		IF NOT fbEcSoERead.bError THEN
			(* read drive diagnostic *)
			fbEcSoERead(
				sNetId		:= stDriveRef.sNetId,
				nSlaveAddr	:= stDriveRef.nSlaveAddr,
				nIdn		:= 375,
				nElement	:= EC_SOE_ELEMENT_VALUE,
				nDriveNo	:= stDriveRef.nDriveNo,
				bCommand	:= FALSE,
				pDstBuf		:= piDiagNumber,
				cbBufLen	:= iSize,
				bExecute	:= FALSE,
				tTimeout	:= tTimeout
			);
			fbEcSoERead(bExecute := TRUE);
			iState	:= 20;
		ELSE
			bBusy	:= FALSE;
			bError	:= TRUE;
			iErrId	:= fbEcSoERead.nErrId;
			MEMSET(piDiagNumber, 0, iSize);
			dwAttribute := 0;
			iState	:= 0;
		END_IF
	END_IF

20: (* wait for read drive diag done *)
	fbEcSoERead(bExecute := FALSE);

	IF NOT fbEcSoERead.bBusy THEN
		fbEcSoERead(bExecute := FALSE);
		iState	:= 0;

		IF NOT fbEcSoERead.bError THEN
			bBusy	:= FALSE;
			(* clear remaining part of array *)
			IF (piDiagNumber^.iActualSize/4 < (iSize-4)/4 ) AND (piDiagNumber^.iMaxSize/4) = (iSize-4)/4 THEN
				FOR I := piDiagNumber^.iActualSize/4 TO (piDiagNumber^.iMaxSize/4) - 1 DO
					piDiagNumber^.arrDiagNumbers[I] := 0;
				END_FOR
			END_IF
		ELSE
			bBusy	:= FALSE;
			bError	:= TRUE;
			iErrId	:= fbEcSoERead.nErrId;
			MEMSET(piDiagNumber, 0, iSize);
		END_IF
	END_IF

END_CASE

bExecute_I := bExecute_I AND bExecute;
END_FUNCTION_BLOCK

(* POU FB_SoEReadMotorTemperature_ByDriveRef, ST *)
FUNCTION_BLOCK FB_SoEReadMotorTemperature_ByDriveRef
VAR_INPUT
	stDriveRef			: ST_DriveRef; 	(* contains sNetID of EcMaster, nSlaveAddr of EcDrive, nDriveNo of EcDrive, either preset or read from NC *)
	bExecute			: BOOL;				(* Function block execution is triggered by a rising edge at this input.*)
	tTimeout			: TIME := DEFAULT_ADS_TIMEOUT;(* States the time before the function is cancelled. *)
END_VAR
VAR_OUTPUT
	bBusy				: BOOL;
	bError				: BOOL;
	iAdsErrId			: UINT;
	iSercosErrId		: UINT;
	dwAttribute			: DWORD;
	fMotorTemperature	: REAL;
END_VAR
{library private}
VAR
	fbEcSoERead 		: FB_EcSoERead;
	iState				: INT;
	bExecute_I			: BOOL;
	iErrId				: UDINT;
	dwData				: ARRAY [0..1] OF DWORD;
	iMotorTemperature	: DINT;
	uiMotorTemperature	: UDINT;

	nFactor				: UINT;					(* bits  0..15 *)
	eLength				: E_SoE_AttribLen;		(* bits 16..18 *)
	eType				: E_SoE_Type;			(* bits 20..22 *)
	nComma				: USINT;				(* bits 24..27 *)
END_VAR
CASE iState OF
0: (* idle *)
	IF bExecute AND NOT bExecute_I THEN
		bExecute_I := bExecute;

		IF NOT bSeqReadDrvAttrAndValue THEN
			(* read Motor Temperature *)
			fbEcSoERead(
				sNetId		:= stDriveRef.sNetId,
				nSlaveAddr	:= stDriveRef.nSlaveAddr,
				nIdn		:= 383,
				nElement	:= 16#44, (* EC_SOE_ELEMENT_VALUE | EC_SOE_ELEMENT_ATTRIBUTE *)
				nDriveNo	:= stDriveRef.nDriveNo,
				bCommand	:= FALSE,
				pDstBuf		:= ADR(dwData),
				cbBufLen	:= SIZEOF(dwData),
				bExecute	:= FALSE,
				tTimeout	:= tTimeout
			);
			iState	:= 10;
		ELSE
			(* read attribute and Motor Temperature sequentially *)
			fbEcSoERead(
				sNetId		:= stDriveRef.sNetId,
				nSlaveAddr	:= stDriveRef.nSlaveAddr,
				nIdn		:= 383,
				nElement	:= EC_SOE_ELEMENT_ATTRIBUTE,
				nDriveNo	:= stDriveRef.nDriveNo,
				bCommand	:= FALSE,
				pDstBuf		:= ADR(dwData[0]),
				cbBufLen	:= SIZEOF(dwData[0]),
				bExecute	:= FALSE,
				tTimeout	:= tTimeout
			);
			iState	:= 5;
		END_IF
		fbEcSoERead(bExecute := TRUE);

		bBusy	:= TRUE;
		bError	:= FALSE;
		iErrId	:= 0;
		iAdsErrId		:= 0;
		iSercosErrId	:= 0;
	END_IF

5: (* wait for read Motor Temperature done *)
	fbEcSoERead(bExecute := FALSE);

	IF NOT fbEcSoERead.bBusy THEN
		fbEcSoERead(bExecute := FALSE);

		IF NOT fbEcSoERead.bError THEN
			(* read attribute and Motor Temperature sequentially *)
			fbEcSoERead(
				sNetId		:= stDriveRef.sNetId,
				nSlaveAddr	:= stDriveRef.nSlaveAddr,
				nIdn		:= 383,
				nElement	:= EC_SOE_ELEMENT_VALUE,
				nDriveNo	:= stDriveRef.nDriveNo,
				bCommand	:= FALSE,
				pDstBuf		:= ADR(dwData[1]),
				cbBufLen	:= SIZEOF(dwData[1]),
				bExecute	:= FALSE,
				tTimeout	:= tTimeout
			);
			fbEcSoERead(bExecute := TRUE);
			iState	:= 10;
		ELSE
			bBusy	:= FALSE;
			bError	:= TRUE;
			iErrId	:= fbEcSoERead.nErrId;
			iAdsErrId		:= UDINT_TO_UINT(iErrId);
			iSercosErrId	:= DWORD_TO_UINT(SHR((UDINT_TO_DWORD(iErrId) AND 16#FFFF0000),16));
			fMotorTemperature := 0;
			iState	:= 0;
		END_IF
	END_IF

10: (* wait for read Motor Temperature done *)
	fbEcSoERead(bExecute := FALSE);

	IF NOT fbEcSoERead.bBusy THEN
		fbEcSoERead(bExecute := FALSE);
		iState	:= 0;

		IF NOT fbEcSoERead.bError THEN
			bBusy	:= FALSE;
			dwAttribute := dwData[0];
			IF (dwAttribute <> 0) THEN
				nFactor	:= DWORD_TO_UINT(dwAttribute          AND 16#0000FFFF); (* bits  0..15 *)
				eLength	:= DWORD_TO_INT(SHR(dwAttribute,  16) AND 16#00000007);	(* bits 16..18 *)
				eType	:= DWORD_TO_INT(SHR(dwAttribute,  20) AND 16#00000007);	(* bits 20..22 *)
				nComma	:= DWORD_TO_USINT(SHR(dwAttribute,24) AND 16#0000000F); (* bits 24..27 *)
			END_IF

			CASE eType OF
			eSoE_Type_UNSIGNED, eSoE_Type_BIN, eSoE_Type_HEX:
				CASE eLength OF
					eSoE_LEN_2BYTE:
						uiMotorTemperature := 0;
						MEMCPY(ADR(uiMotorTemperature), ADR(dwData[1]), UDINT#2);
						fMotorTemperature := UDINT_TO_REAL(uiMotorTemperature) * nFactor / EXPT(10,nComma);
					eSoE_LEN_4BYTE:
						MEMCPY(ADR(uiMotorTemperature), ADR(dwData[1]), UDINT#4);
						fMotorTemperature := UDINT_TO_REAL(uiMotorTemperature) * nFactor / EXPT(10,nComma);
					ELSE
						bError := TRUE;
						iErrId := 16#705; (* parameter size not correct *)
						fMotorTemperature := 0;
				END_CASE

			eSoE_Type_SIGNED:
				CASE eLength OF
					eSoE_LEN_2BYTE:
						iMotorTemperature := 0;
						MEMCPY(ADR(iMotorTemperature), ADR(dwData[1]), UDINT#2);
						fMotorTemperature := DINT_TO_REAL(iMotorTemperature) * nFactor / EXPT(10,nComma);
					eSoE_LEN_4BYTE:
						MEMCPY(ADR(iMotorTemperature), ADR(dwData[1]), UDINT#4);
						fMotorTemperature := DINT_TO_REAL(iMotorTemperature) * nFactor / EXPT(10,nComma);
					ELSE
						bError := TRUE;
						iErrId := 16#705; (* parameter size not correct *)
						fMotorTemperature := 0;
				END_CASE

			ELSE
				bError := TRUE;
				iErrId := 16#706; (* invalid parameter value(s) *)
				fMotorTemperature := 0;
			END_CASE
		ELSE
			bBusy	:= FALSE;
			bError	:= TRUE;
			iErrId	:= fbEcSoERead.nErrId;
			iAdsErrId		:= UDINT_TO_UINT(iErrId);
			iSercosErrId	:= DWORD_TO_UINT(SHR((UDINT_TO_DWORD(iErrId) AND 16#FFFF0000),16));
			fMotorTemperature := 0;
		END_IF
	END_IF

END_CASE

bExecute_I := bExecute_I AND bExecute;
END_FUNCTION_BLOCK

(* POU FB_SoEReset_ByDriveRef, ST *)
FUNCTION_BLOCK FB_SoEReset_ByDriveRef
VAR_INPUT
	stDriveRef		: ST_DriveRef; 	(* contains sNetID of EcMaster, nSlaveAddr of EcDrive, nDriveNo of EcDrive, either preset or read from NC *)
	bExecute		: BOOL;			(* Function block execution is triggered by a rising edge at this input.*)
	tTimeout		: TIME := T#10s;(* States the time before the function is cancelled. (up to 10s) *)
END_VAR
VAR_OUTPUT
	bBusy			: BOOL;
	bError			: BOOL;
	iAdsErrId		: UINT;
	iSercosErrId	: UINT;
END_VAR
{library private}
VAR
	fbEcExecuteCmd	: FB_SoEExecuteCommand_ByDriveRef;
	iState			: INT;
	bExecute_I		: BOOL;
	iReset			: UINT := 3;
END_VAR
CASE iState OF
0: (* idle *)
	IF bExecute AND NOT bExecute_I THEN
		bExecute_I := bExecute;

		(* reset drive *)
		fbEcExecuteCmd(
			stDriveRef	:= stDriveRef,
			nIdn		:= S_0_IDN + 99,
			bExecute	:= FALSE,
			tTimeout	:= tTimeout
		);

		fbEcExecuteCmd(bExecute := TRUE);

		iState	:= 10;
		bBusy	:= TRUE;
		bError	:= FALSE;
		iAdsErrId		:= 0;
		iSercosErrId	:= 0;
	END_IF

10: (* wait for drive reset done *)
	fbEcExecuteCmd(bExecute := FALSE);

	IF NOT fbEcExecuteCmd.bBusy THEN
		fbEcExecuteCmd(bExecute := FALSE);

		IF NOT fbEcExecuteCmd.bError THEN
			(* reset done, drive in OP *)
			iState	:= 0;
			bBusy	:= FALSE;
		ELSE
			iState	:= 0;
			bBusy	:= FALSE;
			bError	:= TRUE;
			iAdsErrId		:= fbEcExecuteCmd.iAdsErrId;
			iSercosErrId	:= fbEcExecuteCmd.iSercosErrId;
		END_IF
	END_IF

END_CASE

bExecute_I := bExecute_I AND bExecute;
END_FUNCTION_BLOCK

(* POU FB_SoEWriteCommandControl_ByDriveRef, ST *)
FUNCTION_BLOCK FB_SoEWriteCommandControl_ByDriveRef
(* The  FB_EcSoEWrite sends a SoE write request to an EtherCAT slave device.*)
VAR_INPUT
	stDriveRef		: ST_DriveRef; 	(* contains sNetID of EcMaster, nSlaveAddr of EcDrive, nDriveNo of EcDrive, either preset or read from NC *)
	nIdn			: WORD;			(* SoE IDN: e.g. "S_0_IDN + 1" for S-0-0001 or "P_0_IDN + 23" for P-0-0023*)
	eCmdControl		: E_SoE_CmdControl;	(* eSoE_CmdControl_Cancel, eSoE_CmdControl_Set, eSoE_CmdControl_SetAndEnable*)
	bExecute		: BOOL;			(* Function block execution is triggered by a rising edge at this input.*)
	tTimeout		: TIME := DEFAULT_ADS_TIMEOUT;(* States the time before the function is cancelled. *)
END_VAR
VAR_OUTPUT
	bBusy			: BOOL;
	bError			: BOOL;
	iAdsErrId		: UINT;
	iSercosErrId	: UINT;
END_VAR
{library private}
VAR
	fbEcSoEWrite	: FB_EcSoEWrite;
	iErrId			: UDINT;
	iState			: INT;
	bExecute_I		: BOOL;
END_VAR
CASE iState OF
0: (* idle *)
	IF bExecute AND NOT bExecute_I THEN
		bExecute_I := bExecute;

		(* write command control *)
		fbEcSoEWrite(
			sNetId		:= stDriveRef.sNetId,
			nSlaveAddr	:= stDriveRef.nSlaveAddr,
			nIdn		:= nIdn,
			nElement	:= EC_SOE_ELEMENT_VALUE,
			nDriveNo	:= stDriveRef.nDriveNo,
			bCommand	:= FALSE,
			pSrcBuf		:= ADR(eCmdControl),
			cbBufLen	:= SIZEOF(eCmdControl),
			bExecute	:= FALSE,
			tTimeout	:= tTimeout
		);
		fbEcSoEWrite(bExecute := TRUE);

		iState	:= 10;
		bBusy	:= TRUE;
		bError	:= FALSE;
		iErrId	:= 0;
		iAdsErrId		:= 0;
		iSercosErrId	:= 0;
	END_IF

10: (* wait for write done *)
	fbEcSoEWrite(bExecute := FALSE);

	IF NOT fbEcSoEWrite.bBusy THEN
		fbEcSoEWrite(bExecute := FALSE);
		iState	:= 0;

		IF NOT fbEcSoEWrite.bError THEN
			bBusy	:= FALSE;
		ELSE
			bBusy	:= FALSE;
			bError	:= TRUE;
			iErrId	:= fbEcSoEWrite.nErrId;
			iAdsErrId		:= UDINT_TO_UINT(iErrId);
			iSercosErrId	:= DWORD_TO_UINT(SHR((UDINT_TO_DWORD(iErrId) AND 16#FFFF0000),16));
		END_IF
	END_IF

END_CASE

bExecute_I := bExecute_I AND bExecute;
END_FUNCTION_BLOCK

(* POU FB_SoEWritePassword_ByDriveRef, ST *)
FUNCTION_BLOCK FB_SoEWritePassword_ByDriveRef
VAR_INPUT
	stDriveRef		: ST_DriveRef; 	(* contains sNetID of EcMaster, nSlaveAddr of EcDrive, nDriveNo of EcDrive, either preset or read from NC *)
	bExecute		: BOOL;			(* Function block execution is triggered by a rising edge at this input.*)
	tTimeout		: TIME := DEFAULT_ADS_TIMEOUT;(* States the time before the function is cancelled. *)
	sPassword		: ST_SoE_String;
END_VAR
VAR_OUTPUT
	bBusy			: BOOL;
	bError			: BOOL;
	iAdsErrId		: UINT;
	iSercosErrId	: UINT;
END_VAR
{library private}
VAR
	fbEcSoEWrite 	: FB_EcSoEWrite;
	iState			: INT;
	bExecute_I		: BOOL;
	iErrId			: UDINT;
END_VAR
CASE iState OF
0: (* idle *)
	IF bExecute AND NOT bExecute_I THEN
		bExecute_I := bExecute;

		sPassword.iMaxSize := LEN(sPassword.strData);
		sPassword.iActualSize := LEN(sPassword.strData);

		(* write drive password *)
		fbEcSoEWrite(
			sNetId		:= stDriveRef.sNetId,
			nSlaveAddr	:= stDriveRef.nSlaveAddr,
			nIdn		:= 267,
			nElement	:= EC_SOE_ELEMENT_VALUE,
			nDriveNo	:= stDriveRef.nDriveNo,
			bCommand	:= FALSE,
			pSrcBuf		:= ADR(sPassword),
			cbBufLen	:= sPassword.iActualSize + 4 + SEL( (UINT_TO_WORD(sPassword.iMaxSize) AND 16#0001) = 16#0001, 0,  1 ),
			bExecute	:= FALSE,
			tTimeout	:= tTimeout
		);
		fbEcSoEWrite(bExecute := TRUE);

		iState	:= 10;
		bBusy	:= TRUE;
		bError	:= FALSE;
		iErrId	:= 0;
		iAdsErrId		:= 0;
		iSercosErrId	:= 0;
	END_IF

10: (* wait for write drive password done *)
	fbEcSoEWrite(bExecute := FALSE);

	IF NOT fbEcSoEWrite.bBusy THEN
		fbEcSoEWrite(bExecute := FALSE);
		iState	:= 0;

		IF NOT fbEcSoEWrite.bError THEN
			bBusy	:= FALSE;
		ELSE
			bBusy	:= FALSE;
			bError	:= TRUE;
			iErrId	:= fbEcSoEWrite.nErrId;
			iAdsErrId		:= UDINT_TO_UINT(iErrId);
			iSercosErrId	:= DWORD_TO_UINT(SHR((UDINT_TO_DWORD(iErrId) AND 16#FFFF0000),16));
		END_IF
	END_IF

END_CASE

bExecute_I := bExecute_I AND bExecute;
END_FUNCTION_BLOCK
